// TIA Portal V17 export
// export: Created 2023-05-07T12:12:22.6228362Z, ExportSetting WithDefaults, DisplayName Totally Integrated Automation Portal, DisplayVersion V17, DisplayName TIA Portal Openness, DisplayVersion V17, DisplayName TIA Portal Version Control Interface, DisplayVersion V17, DisplayName TIA Portal Test Suite Advanced, DisplayVersion V17, DisplayName STEP 7 Professional, DisplayVersion V17, DisplayName SIMATIC Energy Suite, DisplayVersion V17, DisplayName STEP 7 Safety, DisplayVersion V17, DisplayName WinCC Professional, DisplayVersion V17
DATA_BLOCK "RandomDisturbance_DB"   // DB5
VERSION : 0.1
// stored: AutoNumber true, InstanceOfName RandomDisturbance, InstanceOfType FB
"RandomDisturbance"
   // VAR_INPUT
   //    DistribanceMode : Int;
   //    Outflow : Int;
   // END_VAR
   // VAR_OUTPUT
   //    DischargeValve : Int;
   // END_VAR
   // VAR
   //    TON_1 { ExternalAccessible := 'False'; ExternalVisible := 'False'; ExternalWritable := 'False'} : TON_TIME;
   //    TON_2 { ExternalAccessible := 'False'; ExternalVisible := 'False'; ExternalWritable := 'False'} : TON_TIME;
   //    TP { ExternalAccessible := 'False'; ExternalVisible := 'False'; ExternalWritable := 'False'} : TP_TIME;
   //    TON_3 { ExternalAccessible := 'False'; ExternalVisible := 'False'; ExternalWritable := 'False'} : TON_TIME;
   //    random { S7_SetPoint := 'True'} : Int;
   //    p_Q : Bool;
   // END_VAR
BEGIN
END_DATA_BLOCK
